(*			
	EVERDE sp. z o.o.
	Rafał Osajda		08.08.2025		TC 4024.66
	Interfejs do wyciągania z SPM przez HMI danych do wyświetlania - dla ramki głównej tryb pracy mycie
*)
INTERFACE ITF_SPM_HMI_00_04_Lacznik EXTENDS  B_Baza.ITF_ZrodloIdentyfikacji

END_INTERFACE

(* stored: Version 1.1.0.1
   Itf ITF_SPM_HMI_00_04_Lacznik: Id {54bd6603-ac92-0fca-279c-5136a5707603} *)
